Fanuc KAREL source: KC00042.KL

PROGRAM KC00042
%NOLOCKGROUP
%ENVIRONMENT REGOPE
VAR
  I: INTEGER
  J: INTEGER
  K: INTEGER
  R: REAL
  B: BOOLEAN
  S: STRING[80]
  T: STRING[80]
  P: PATH
  Q: PATH
  AI: ARRAY[8] OF INTEGER
  AB: ARRAY[244] OF BYTE
  JP: JOINTPOS
BEGIN
  JP = GET_TPE_JPOS_REG(I,J)
END KC00042
